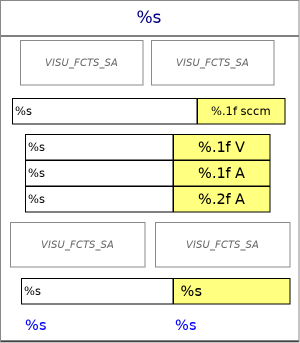
VISUALIZATION SA_IAD  // 300x343
VAR_IN_OUT
	m_Input_CANON_ION : BLOCK_CANON_ION_MARK3;
	m_Input_IAD : BLOCK_MARK3_PLUS;
END_VAR
    Rectangle (-1,-2 300x343)
    Rectangle (25,134 148x26), "%s", text list: 'TextList_IAD', text index: 0
    Rectangle (173,134 97x26), "%.1f V", text variable: m_Input_IAD.PRM_ANODE_VOLTAGE, input disabled if: ((NOT PRG_User.ACTU_USER.MAINTENANCE AND NOT PRG_User.ACTU_USER.FONCTION_SA AND NOT PRG_User.ACTU_USER.MODIF_ENLIGNE) OR (NOT MACHINE.STATE_Wait_Prod AND NOT MACHINE.STATE_Manu)) <> 0
        OnMouseDown: write the text variable via VisuDialogs.Numpad, min 0, max 300
    Rectangle (21,278 152x26), "%s", text list: 'TextList_IAD', text index: 11
    Rectangle (173,278 117x26), "%s", text variable: m_Input_CANON_ION.PRM_TPS_IAD, input disabled if: ((NOT PRG_User.ACTU_USER.MAINTENANCE AND NOT PRG_User.ACTU_USER.FONCTION_SA AND NOT PRG_User.ACTU_USER.MODIF_ENLIGNE) OR (NOT MACHINE.STATE_Wait_Prod AND NOT MACHINE.STATE_Manu)) <> 0
        OnMouseDown: write the text variable via VisuDialogs.Keypad
    Rectangle (172,312 117x26), "%s", text variable: m_Input_CANON_ION.STATE_IAD, invisible if: NOT m_Input_CANON_ION.OP_IAD.Etape.3
    Rectangle (25,186 148x26), "%s", text list: 'TextList_IAD', text index: 2
    Rectangle (173,186 97x26), "%.2f A", text variable: m_Input_IAD.PRM_NEUTRAL_CURRENT, input disabled if: ((NOT PRG_User.ACTU_USER.MAINTENANCE AND NOT PRG_User.ACTU_USER.FONCTION_SA AND NOT PRG_User.ACTU_USER.MODIF_ENLIGNE) OR (NOT MACHINE.STATE_Wait_Prod AND NOT MACHINE.STATE_Manu)) <> 0
        OnMouseDown: write the text variable via VisuDialogs.Numpad, min 0, max 1.86
    Rectangle (25,160 148x26), "%s", text list: 'TextList_IAD', text index: 1
    Rectangle (173,160 97x26), "%.1f A", text variable: m_Input_IAD.PRM_ANODE_CURRENT, input disabled if: ((NOT PRG_User.ACTU_USER.MAINTENANCE AND NOT PRG_User.ACTU_USER.FONCTION_SA AND NOT PRG_User.ACTU_USER.MODIF_ENLIGNE) OR (NOT MACHINE.STATE_Wait_Prod AND NOT MACHINE.STATE_Manu)) <> 0
        OnMouseDown: write the text variable via VisuDialogs.Numpad, min 0, max 15
    Rectangle (-1,-2 300x38), "%s", text list: 'TextList_IAD', text index: 10
    Rectangle (22,312 147x26), "%s", invisible if: NOT m_Input_CANON_ION.OP_IAD.Etape.3, text list: 'TextList_IAD'
    Rectangle (12,98 185x26), "%s", text list: 'TextList_IAD', text index: 8
    Rectangle (197,98 88x26), "%.1f sccm", text variable: m_Input_CANON_ION.PRM_GAZ_1C_AMORCAGE, input disabled if: ((NOT PRG_User.ACTU_USER.MAINTENANCE AND NOT PRG_User.ACTU_USER.FONCTION_SA AND NOT PRG_User.ACTU_USER.MODIF_ENLIGNE) OR (NOT MACHINE.STATE_Wait_Prod AND NOT MACHINE.STATE_Manu)) <> 0
        OnMouseDown: write the text variable via VisuDialogs.Numpad, min 0, max 100
    Frame (151,40 123x45)
        shows VISU_FCTS_SA(m_Input_ID_XML := 7, m_Input_UserRight := PRG_USER.ACTU_USER.FONCTION_SA, m_Input_Operation := m_Input_CANON_ION.OP_ARRET)
    Frame (20,40 123x45)
        shows VISU_FCTS_SA(m_Input_ID_XML := 5, m_Input_UserRight := PRG_USER.ACTU_USER.FONCTION_SA, m_Input_Operation := m_Input_CANON_ION.OP_MARCHE)
    Frame (155,222 135x45)
        shows VISU_FCTS_SA(m_Input_ID_XML := 27, m_Input_UserRight := PRG_USER.ACTU_USER.FONCTION_SA, m_Input_Operation := m_Input_CANON_ION.OP_STOP_IAD)
    Frame (10,222 135x45)
        shows VISU_FCTS_SA(m_Input_ID_XML := 26, m_Input_UserRight := PRG_USER.ACTU_USER.FONCTION_SA, m_Input_Operation := m_Input_CANON_ION.OP_IAD)
END_VISUALIZATION

(* stored: Version 1.1.0.1, ProductVersion 3.1.4024.10
   Visu SA_IAD: Id {aae97bdb-a92f-4308-94e7-26941fe25cfa} *)
